// SIMATIC S7-200 project (STEP 7-Micro/WIN), CPU 222 REL 02.01

SYMBOL_TABLE USER1
E0               M0.0     // ETAPA 0
E1               M0.1     // ETAPA 1
E2               M0.2     // ETAPA 2
E3               M0.3     // ETAPA 3
E10              M1.0     // ETAPA 10
E11              M1.1     // ETAPA 11
E12              M1.2     // ETAPA 12
SCP              I0.6     // SENSOR CAIXA PEQUENA
CONT1            C0       // PRIMEIRO CONTADOR DE 5
SCG              I0.7     // SENSOR CAIXA GRANDE
CONT2            C1       // SEGUNDO CONTADOR DE 8
E13              M1.3     // ETAPA 13
EST1             Q0.0     // ESTEIRA 1
EST2             Q0.1     // ESTEIRA 2
CP               Q0.2     // SAIDA DE CAIXAS PEQUENAS
CG               Q0.3     // SAIDA DE CAIXAS GRANDES
END_SYMBOL_TABLE

ORGANIZATION_BLOCK MAIN:OB1
TITLE=PROGRAM COMMENTS
BEGIN
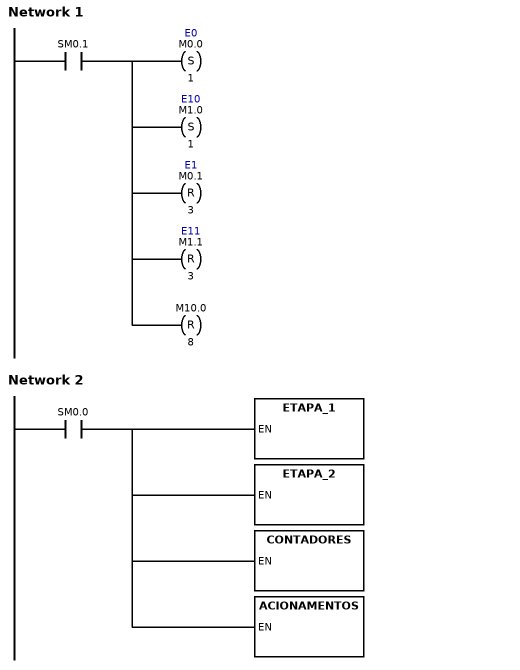
Network 1
LD     SM0.1
S      E0:M0.0, 1
S      E10:M1.0, 1
R      E1:M0.1, 3
R      E11:M1.1, 3
R      M10.0, 8
Network 2
LD     SM0.0
CALL   ETAPA_1:SBR0
CALL   ETAPA_2:SBR1
CALL   CONTADORES:SBR2
CALL   ACIONAMENTOS:SBR3
END_ORGANIZATION_BLOCK

SUBROUTINE_BLOCK ETAPA_1:SBR0
TITLE=SUBROUTINE COMMENTS
BEGIN
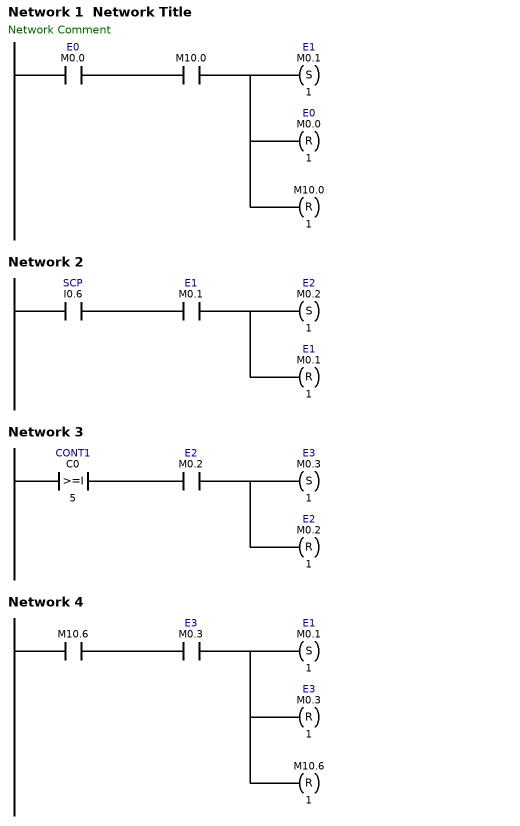
Network 1 // Network Title
// Network Comment
LD     E0:M0.0
A      M10.0
S      E1:M0.1, 1
R      E0:M0.0, 1
R      M10.0, 1
Network 2
LD     SCP:I0.6
A      E1:M0.1
S      E2:M0.2, 1
R      E1:M0.1, 1
Network 3
LDW>=  CONT1:C0, 5
A      E2:M0.2
S      E3:M0.3, 1
R      E2:M0.2, 1
Network 4
LD     M10.6
A      E3:M0.3
S      E1:M0.1, 1
R      E3:M0.3, 1
R      M10.6, 1
END_SUBROUTINE_BLOCK

SUBROUTINE_BLOCK ETAPA_2:SBR1
TITLE=SUBROUTINE COMMENTS
BEGIN
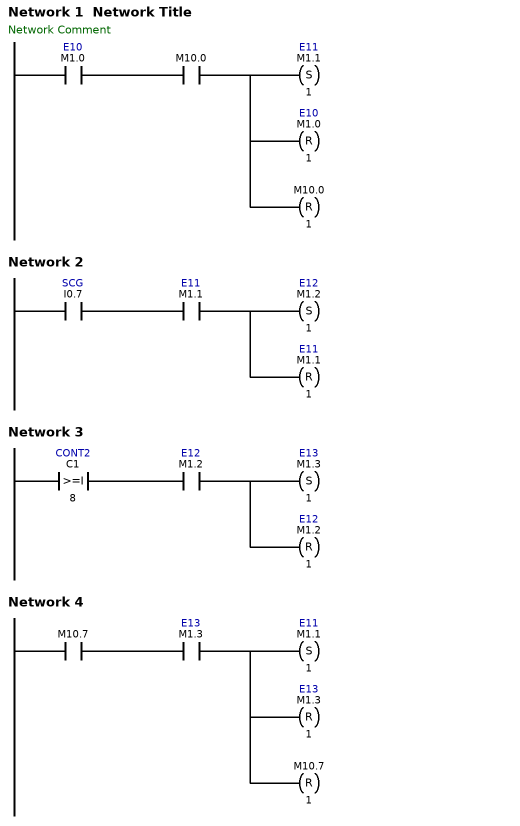
Network 1 // Network Title
// Network Comment
LD     E10:M1.0
A      M10.0
S      E11:M1.1, 1
R      E10:M1.0, 1
R      M10.0, 1
Network 2
LD     SCG:I0.7
A      E11:M1.1
S      E12:M1.2, 1
R      E11:M1.1, 1
Network 3
LDW>=  CONT2:C1, 8
A      E12:M1.2
S      E13:M1.3, 1
R      E12:M1.2, 1
Network 4
LD     M10.7
A      E13:M1.3
S      E11:M1.1, 1
R      E13:M1.3, 1
R      M10.7, 1
END_SUBROUTINE_BLOCK

SUBROUTINE_BLOCK CONTADORES:SBR2
TITLE=SUBROUTINE COMMENTS
BEGIN
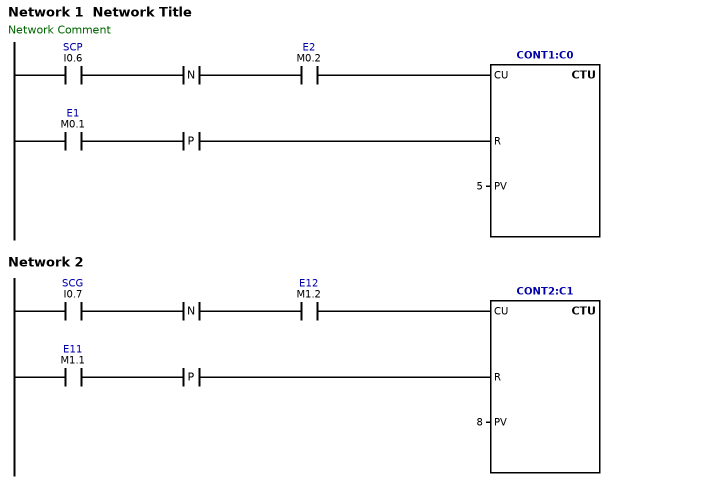
Network 1 // Network Title
// Network Comment
LD     SCP:I0.6
ED
A      E2:M0.2
LD     E1:M0.1
EU
CTU    CONT1:C0, 5
Network 2
LD     SCG:I0.7
ED
A      E12:M1.2
LD     E11:M1.1
EU
CTU    CONT2:C1, 8
END_SUBROUTINE_BLOCK

SUBROUTINE_BLOCK ACIONAMENTOS:SBR3
TITLE=SUBROUTINE COMMENTS
BEGIN
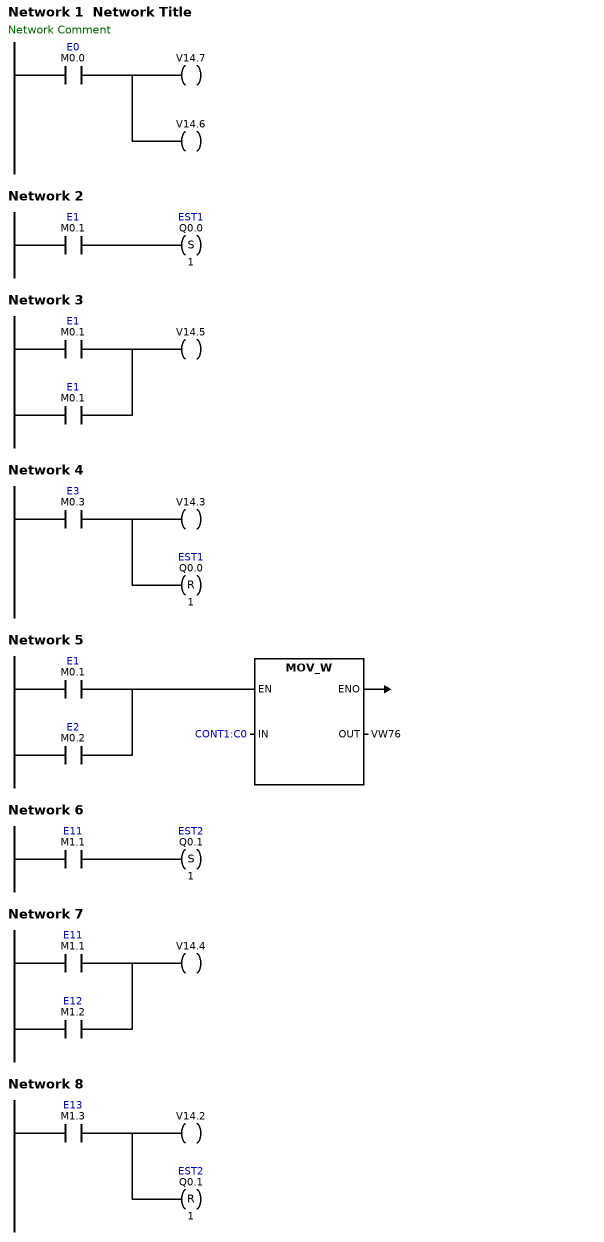
Network 1 // Network Title
// Network Comment
LD     E0:M0.0
=      V14.7
=      V14.6
Network 2
LD     E1:M0.1
S      EST1:Q0.0, 1
Network 3
LD     E1:M0.1
O      E1:M0.1
=      V14.5
Network 4
LD     E3:M0.3
=      V14.3
R      EST1:Q0.0, 1
Network 5
LD     E1:M0.1
O      E2:M0.2
MOVW   CONT1:C0, VW76
Network 6
LD     E11:M1.1
S      EST2:Q0.1, 1
Network 7
LD     E11:M1.1
O      E12:M1.2
=      V14.4
Network 8
LD     E13:M1.3
=      V14.2
R      EST2:Q0.1, 1
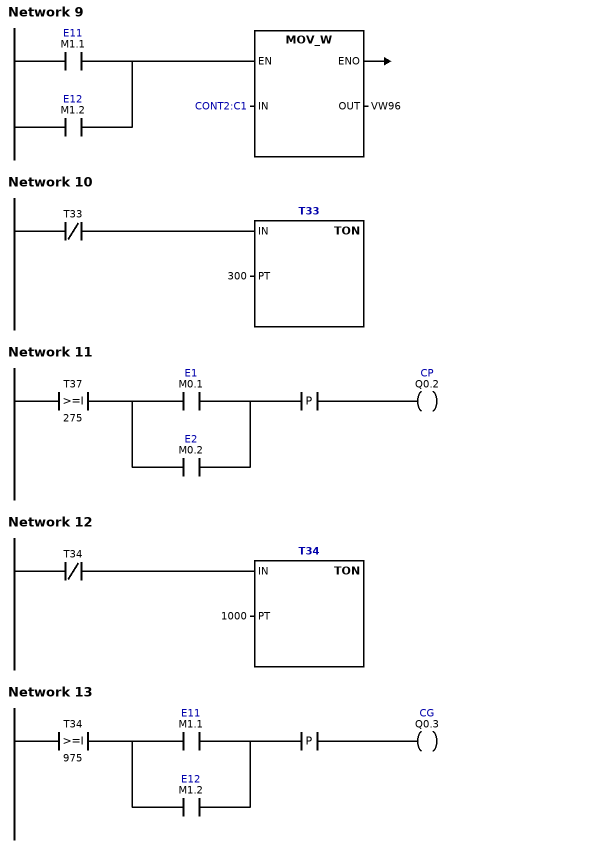
Network 9
LD     E11:M1.1
O      E12:M1.2
MOVW   CONT2:C1, VW96
Network 10
LDN    T33
TON    T33, 300
Network 11
LDW>=  T37, 275
LD     E1:M0.1
O      E2:M0.2
ALD
EU
=      CP:Q0.2
Network 12
LDN    T34
TON    T34, 1000
Network 13
LDW>=  T34, 975
LD     E11:M1.1
O      E12:M1.2
ALD
EU
=      CG:Q0.3
END_SUBROUTINE_BLOCK

DATA_BLOCK_TAB TD_DATA_0
BEGIN
VB0      'TD'
VB2      16#10               //Set Language to English, set Update to as fast as possible 
VB3      16#80               //Set the display to 20 character mode; Enter key V3.1; Up key V3.2; Down key V3.3;
VB4      6                   //Set the number of messages
VB5      16#A                //Set the Function Keys notification bits to M10.0 - M10.7, F-Keys configured to set M-bits
VW6      24                  //Set the starting address for messages to  VB24
VW8      14                  //Set the starting address for message enable bits to VB14
VW10     65535               //Global Password (if enabled)
VW12     2                   //Character Set = Latin 1 (Bold)
//MESSAGE 1
//Message Enable Bit V14.7 
VB24     ' PARTIDA ==> F1     '
//MESSAGE 2
//Message Enable Bit V14.6 
VB44     '                    '
//MESSAGE 3
//Message Enable Bit V14.5 
VB64     'LOTE1 ON  '
VB74     16#0                //No Edit;No Acknowledgement;No Password;
VB75     16#30               //Unsigned Word; 0 Digits to the right of the decimal;
VW76     16#0                //Embedded Data Value: Move data for display here.
VB78     ' PEÇAS'
//MESSAGE 4
//Message Enable Bit V14.4 
VB84     'LOTE2 ON  '
VB94     16#0                //No Edit;No Acknowledgement;No Password;
VB95     16#30               //Unsigned Word; 0 Digits to the right of the decimal;
VW96     16#0                //Embedded Data Value: Move data for display here.
VB98     ' PEÇAS'
//MESSAGE 5
//Message Enable Bit V14.3 
VB104    'L1=OK  CONTINUAR=>F7'
//MESSAGE 6
//Message Enable Bit V14.2 
VB124    'L2=OK  CONTINUAR=>F8'
//END TD200_BLOCK ------------------------------
//DATA PAGE COMMENTS
//Press F1 for help and example data page
END_DATA_BLOCK_TAB
